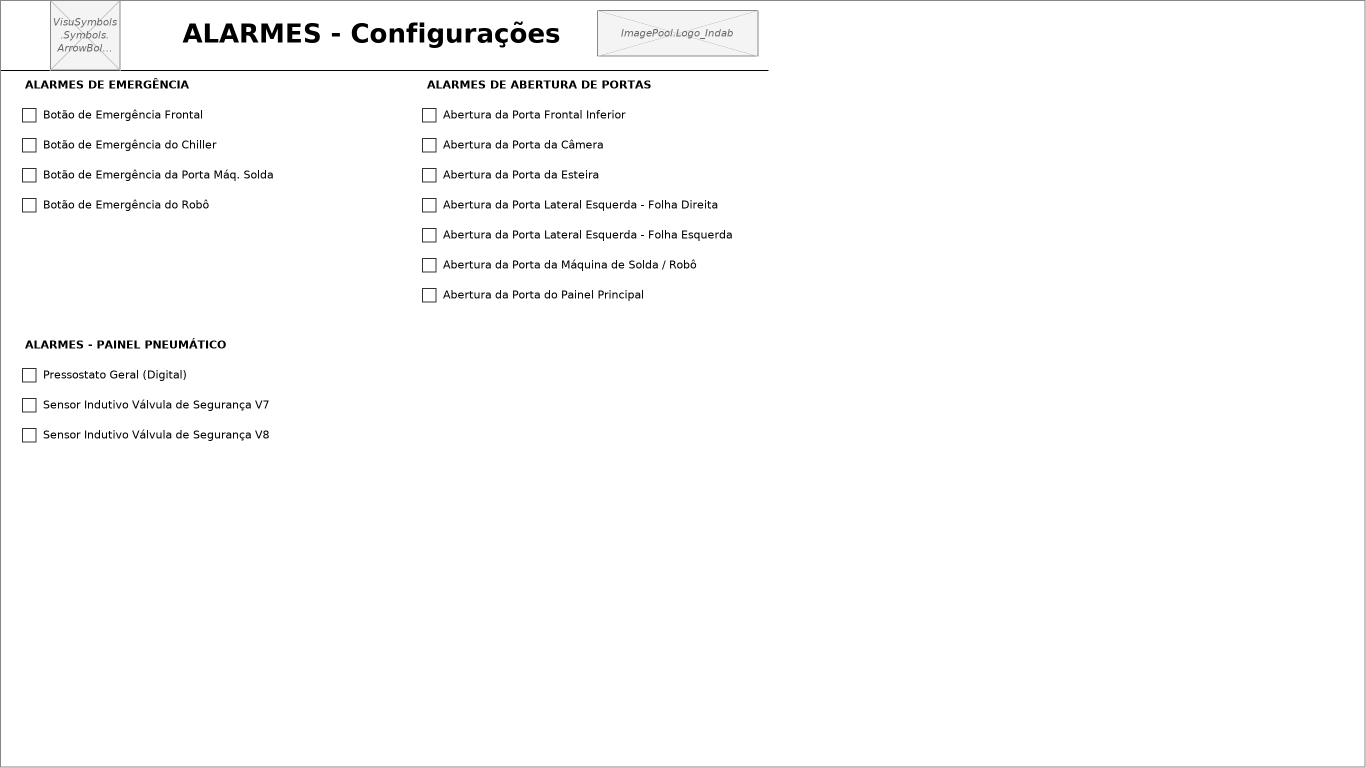
VISUALIZATION Tela_Alarmes_2  // 1366x768
    Line (0,70) (768,70)
    Line (0,1312) (768,1312)
    Image (597,10 161x46), image: ImagePool.Logo_Indab
    Rectangle (584,1340 180x24), "%t[dd/MM/yyyy]"
    Rectangle (584,1316 180x24), "%t[HH:mm:ss]"
    Label (153,7 437x53), "ALARMES - Configurações"
    Button (15,1315 175x45), "RECEITAS"
        OnMouseClick: change screen: Tela_Receita
    Checkbox (420,190 313x30), "Abertura da Porta Lateral Esquerda - Folha Direita"
    Checkbox (420,220 329x30), "Abertura da Porta Lateral Esquerda - Folha Esquerda"
    Checkbox (420,250 296x30), "Abertura da Porta da Máquina de Solda / Robô"
    Rectangle (22,75 237x20), "ALARMES DE EMERGÊNCIA"
    Rectangle (424,75 237x20), "ALARMES DE ABERTURA DE PORTAS"
    Checkbox (20,100 200x30), "Botão de Emergência Frontal"
    Checkbox (20,130 214x30), "Botão de Emergência do Chiller"
    Checkbox (20,160 278x30), "Botão de Emergência da Porta Máq. Solda"
    Checkbox (20,190 220x30), "Botão de Emergência do Robô"
    Checkbox (420,100 238x30), "Abertura da Porta Frontal Inferior"
    Checkbox (420,130 200x30), "Abertura da Porta da Câmera"
    Checkbox (420,160 200x30), "Abertura da Porta da Esteira"
    Checkbox (420,280 243x30), "Abertura da Porta do Painel Principal"
    Rectangle (22,335 237x20), "ALARMES - PAINEL PNEUMÁTICO"
    Checkbox (20,360 200x30), "Pressostato Geral (Digital)"
    Checkbox (20,390 286x30), "Sensor Indutivo Válvula de Segurança V7"
    Checkbox (20,420 278x30), "Sensor Indutivo Válvula de Segurança V8"
    Image (50,0 70x70), image: VisuSymbols.Symbols.ArrowBoldLeft
        OnMouseClick: change screen: Tela_Alarmes_1
    Button (375,1315 175x45), "PRODUÇÃO"
        OnMouseClick: change screen: Tela_Producao
    Button (195,1315 175x45), "MANUTENÇÃO"
        OnMouseClick: change screen: Tela_Manutencao
END_VISUALIZATION

(* stored: Version 1.1.0.1, ProductVersion 3.1.4024.11
   Visu Tela_Alarmes_2: Id {4069a176-e753-4986-9627-08977c767163} *)
